// TIA Portal V16 export
// export: Created 2023-03-29T11:03:24.7291018Z, ExportSetting WithDefaults, DisplayName Totally Integrated Automation Portal, DisplayVersion V16 Update 6, DisplayName TIA Portal Version Control Interface, DisplayVersion V16 Update 2, DisplayName TIA Portal Openness, DisplayVersion V16 Update 6, DisplayName STEP 7 Professional, DisplayVersion V16 Update 6, DisplayName STEP 7 Safety, DisplayVersion V16, DisplayName WinCC Advanced, DisplayVersion V16 Update 6
FUNCTION_BLOCK "Client_ModbusTCP_sending_analogs"   // FB4, LAD
TITLE = Wysyłanie analogów
{ S7_Optimized_Access := 'TRUE' }
AUTHOR : rtecmer
VERSION : 0.1
// Wysyłanie pomiarów
// stored: AutoNumber true, IsIECCheckEnabled false, IsRetainMemResEnabled false, MemoryReserve 250, SetENOAutomatically false, UDAEnableTagReadback false
   VAR_IN_OUT
      modbustcp_przetwarzanie_in : Bool;
      modbustcp_przetwarzanie_out : Bool;
   END_VAR
   VAR_TEMP   // added for the SCL form of the ladder/FBD networks
      _w1 : Bool;
      _w2 : Bool;
   END_VAR
BEGIN

REGION Network 2: Inicjacja modbus po błędzie i restarcie
END_REGION

REGION Network 3
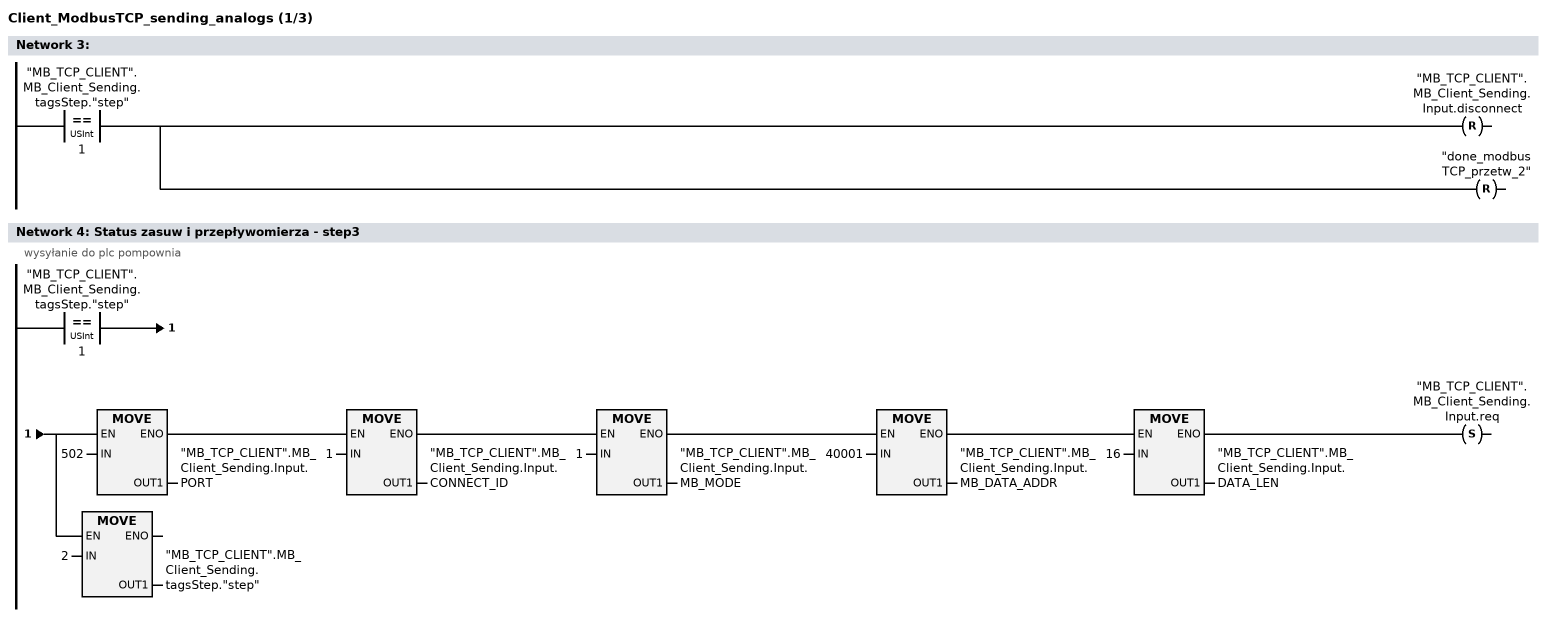
   RUNG wire#powerrail
      { S7_Templates := "SrcType := USInt" } EQ_Contact(in1 := "MB_TCP_CLIENT".MB_Client_Sending.tagsStep."step", in2 := 1)
      wire#w1
      R_Coil( "MB_TCP_CLIENT".MB_Client_Sending.Input.disconnect )
   END_RUNG
   RUNG wire#w1
      R_Coil( "done_modbusTCP_przetw_2" )
   END_RUNG
   // the same network as SCL:
   IF "MB_TCP_CLIENT".MB_Client_Sending.tagsStep."step" = 1 THEN
       "MB_TCP_CLIENT".MB_Client_Sending.Input.disconnect := FALSE;
       "done_modbusTCP_przetw_2" := FALSE;
   END_IF;
END_REGION

REGION Network 4: Status zasuw i przepływomierza - step3
   // wysyłanie do plc pompownia
   RUNG wire#powerrail
      { S7_Templates := "SrcType := USInt" } EQ_Contact(in1 := "MB_TCP_CLIENT".MB_Client_Sending.tagsStep."step", in2 := 1)
      wire#w1
      { S7_GenerateENO := "TRUE" } Move(in := 502, out1 => "MB_TCP_CLIENT".MB_Client_Sending.Input.PORT)
      { S7_GenerateENO := "TRUE" } Move(in := 1, out1 => "MB_TCP_CLIENT".MB_Client_Sending.Input.CONNECT_ID)
      { S7_GenerateENO := "TRUE" } Move(in := 1, out1 => "MB_TCP_CLIENT".MB_Client_Sending.Input.MB_MODE)
      { S7_GenerateENO := "TRUE" } Move(in := 40001, out1 => "MB_TCP_CLIENT".MB_Client_Sending.Input.MB_DATA_ADDR)
      { S7_GenerateENO := "TRUE" } Move(in := 16, out1 => "MB_TCP_CLIENT".MB_Client_Sending.Input.DATA_LEN)
      S_Coil( "MB_TCP_CLIENT".MB_Client_Sending.Input.req )
   END_RUNG
   RUNG wire#w1
      { S7_GenerateENO := "TRUE" } Move(in := 2, out1 => "MB_TCP_CLIENT".MB_Client_Sending.tagsStep."step")
   END_RUNG
   // the same network as SCL:
   // ENO of a box is taken as its EN; it also drops when the box reports an error
   IF "MB_TCP_CLIENT".MB_Client_Sending.tagsStep."step" = 1 THEN
       "MB_TCP_CLIENT".MB_Client_Sending.Input.PORT := 502;
       "MB_TCP_CLIENT".MB_Client_Sending.Input.CONNECT_ID := 1;
       "MB_TCP_CLIENT".MB_Client_Sending.Input.MB_MODE := 1;
       "MB_TCP_CLIENT".MB_Client_Sending.Input.MB_DATA_ADDR := 40001;
       "MB_TCP_CLIENT".MB_Client_Sending.Input.DATA_LEN := 16;
       "MB_TCP_CLIENT".MB_Client_Sending.Input.req := TRUE;
       "MB_TCP_CLIENT".MB_Client_Sending.tagsStep."step" := 2;
   END_IF;
END_REGION

REGION Network 5: step 3
   // Analogi
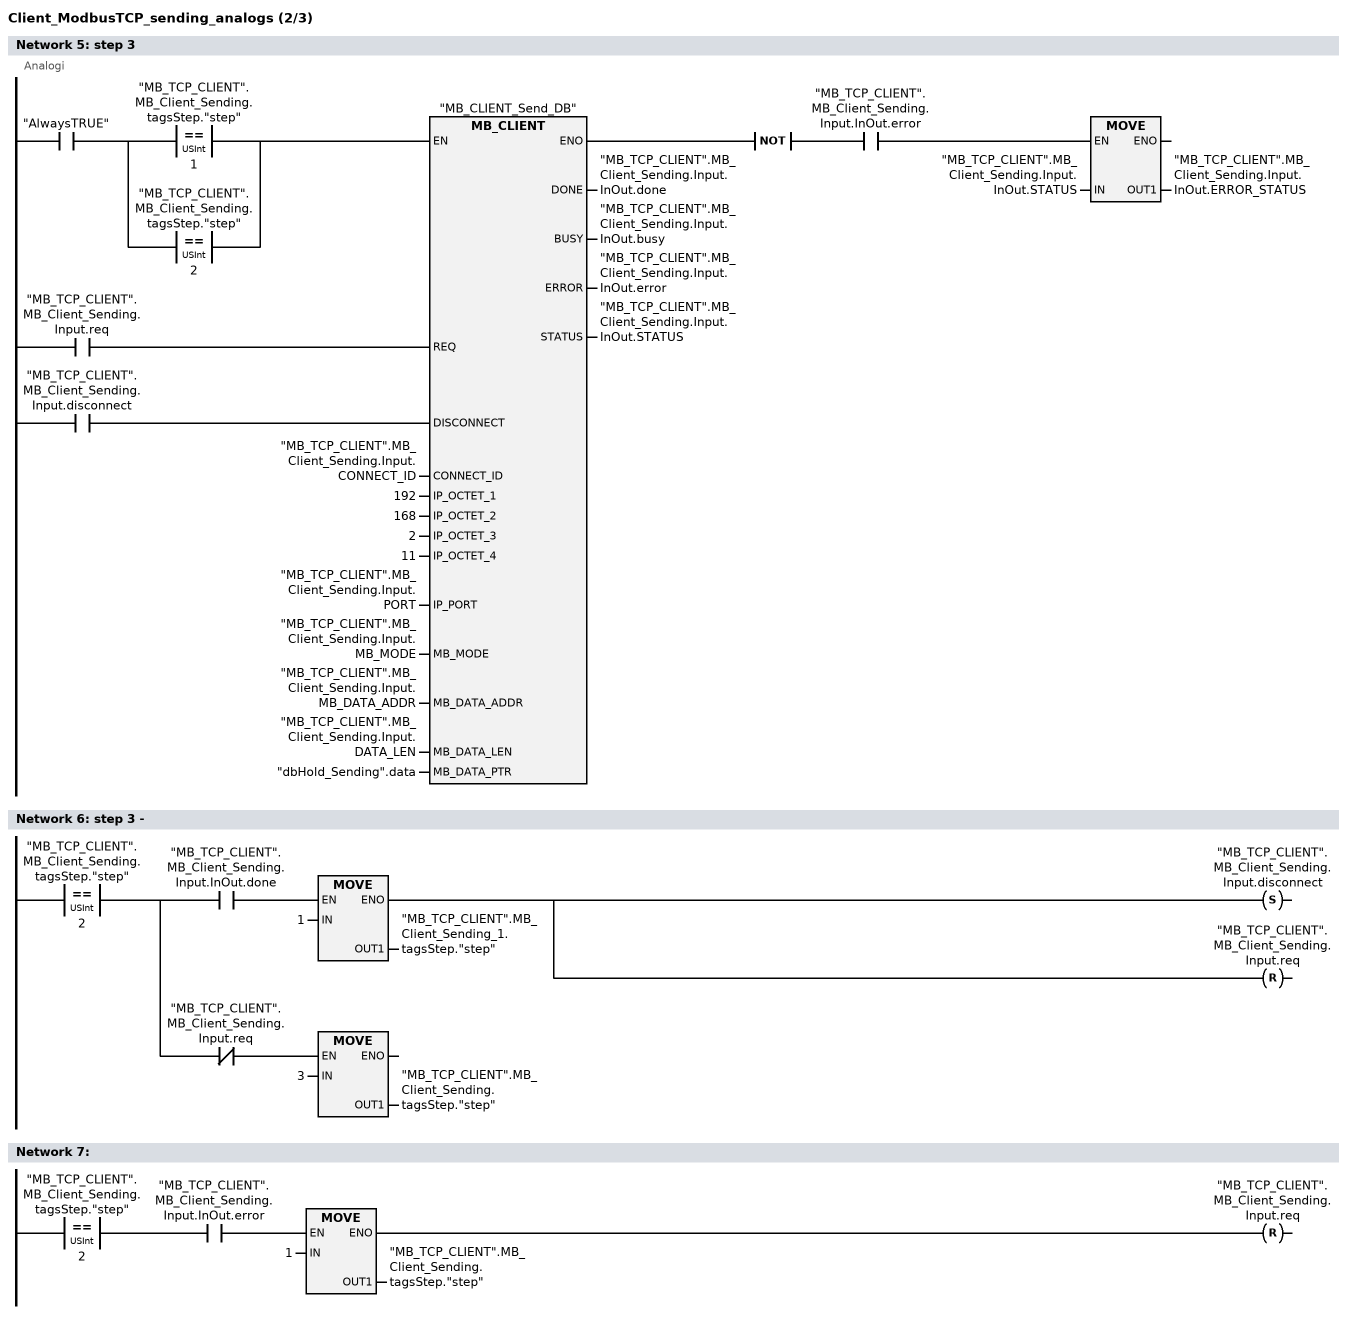
   RUNG wire#powerrail
      Contact( "AlwaysTRUE" )
      wire#w1
      { S7_Templates := "SrcType := USInt" } EQ_Contact(in1 := "MB_TCP_CLIENT".MB_Client_Sending.tagsStep."step", in2 := 1)
      wire#w2
      { S7_Templates := "[card1200 := 1, card1500 := 0]" } "MB_CLIENT_Send_DB".MB_CLIENT(REQ := wire#w3, DISCONNECT := wire#w4, CONNECT_ID := "MB_TCP_CLIENT".MB_Client_Sending.Input.CONNECT_ID, IP_OCTET_1 := 192, IP_OCTET_2 := 168, IP_OCTET_3 := 2, IP_OCTET_4 := 11, IP_PORT := "MB_TCP_CLIENT".MB_Client_Sending.Input.PORT, MB_MODE := "MB_TCP_CLIENT".MB_Client_Sending.Input.MB_MODE, MB_DATA_ADDR := "MB_TCP_CLIENT".MB_Client_Sending.Input.MB_DATA_ADDR, MB_DATA_LEN := "MB_TCP_CLIENT".MB_Client_Sending.Input.DATA_LEN, MB_DATA_PTR := "dbHold_Sending".data, DONE => "MB_TCP_CLIENT".MB_Client_Sending.Input.InOut.done, BUSY => "MB_TCP_CLIENT".MB_Client_Sending.Input.InOut.busy, ERROR => "MB_TCP_CLIENT".MB_Client_Sending.Input.InOut.error, STATUS => "MB_TCP_CLIENT".MB_Client_Sending.Input.InOut.STATUS)
      Not()
      Contact( "MB_TCP_CLIENT".MB_Client_Sending.Input.InOut.error )
      Move(in := "MB_TCP_CLIENT".MB_Client_Sending.Input.InOut.STATUS, out1 => "MB_TCP_CLIENT".MB_Client_Sending.Input.InOut.ERROR_STATUS)
   END_RUNG
   RUNG wire#w1
      { S7_Templates := "SrcType := USInt" } EQ_Contact(in1 := "MB_TCP_CLIENT".MB_Client_Sending.tagsStep."step", in2 := 2)
   END_RUNG wire#w2
   RUNG wire#powerrail
      Contact( "MB_TCP_CLIENT".MB_Client_Sending.Input.req )
   END_RUNG wire#w3
   RUNG wire#powerrail
      Contact( "MB_TCP_CLIENT".MB_Client_Sending.Input.disconnect )
   END_RUNG wire#w4
   // the same network as SCL:
   #_w1 := "AlwaysTRUE" AND (("MB_TCP_CLIENT".MB_Client_Sending.tagsStep."step" = 1) OR ("MB_TCP_CLIENT".MB_Client_Sending.tagsStep."step" = 2));
   "MB_CLIENT_Send_DB"(EN := #_w1,   // MB_CLIENT
                       REQ := "MB_TCP_CLIENT".MB_Client_Sending.Input.req,
                       DISCONNECT := "MB_TCP_CLIENT".MB_Client_Sending.Input.disconnect,
                       CONNECT_ID := "MB_TCP_CLIENT".MB_Client_Sending.Input.CONNECT_ID,
                       IP_OCTET_1 := 192,
                       IP_OCTET_2 := 168,
                       IP_OCTET_3 := 2,
                       IP_OCTET_4 := 11,
                       IP_PORT := "MB_TCP_CLIENT".MB_Client_Sending.Input.PORT,
                       MB_MODE := "MB_TCP_CLIENT".MB_Client_Sending.Input.MB_MODE,
                       MB_DATA_ADDR := "MB_TCP_CLIENT".MB_Client_Sending.Input.MB_DATA_ADDR,
                       MB_DATA_LEN := "MB_TCP_CLIENT".MB_Client_Sending.Input.DATA_LEN,
                       MB_DATA_PTR := "dbHold_Sending".data,
                       DONE => "MB_TCP_CLIENT".MB_Client_Sending.Input.InOut.done,
                       BUSY => "MB_TCP_CLIENT".MB_Client_Sending.Input.InOut.busy,
                       ERROR => "MB_TCP_CLIENT".MB_Client_Sending.Input.InOut.error,
                       STATUS => "MB_TCP_CLIENT".MB_Client_Sending.Input.InOut.STATUS,
                       ENO => #_w2);
   IF NOT #_w2 AND "MB_TCP_CLIENT".MB_Client_Sending.Input.InOut.error THEN
       "MB_TCP_CLIENT".MB_Client_Sending.Input.InOut.ERROR_STATUS := "MB_TCP_CLIENT".MB_Client_Sending.Input.InOut.STATUS;
   END_IF;
END_REGION

REGION Network 6: step 3 -
   RUNG wire#powerrail
      { S7_Templates := "SrcType := USInt" } EQ_Contact(in1 := "MB_TCP_CLIENT".MB_Client_Sending.tagsStep."step", in2 := 2)
      wire#w1
      Contact( "MB_TCP_CLIENT".MB_Client_Sending.Input.InOut.done )
      Move(in := 1, out1 => "MB_TCP_CLIENT".MB_Client_Sending_1.tagsStep."step")
      wire#w2
      S_Coil( "MB_TCP_CLIENT".MB_Client_Sending.Input.disconnect )
   END_RUNG
   RUNG wire#w2
      R_Coil( "MB_TCP_CLIENT".MB_Client_Sending.Input.req )
   END_RUNG
   RUNG wire#w1
      I_Contact( "MB_TCP_CLIENT".MB_Client_Sending.Input.req )
      Move(in := 3, out1 => "MB_TCP_CLIENT".MB_Client_Sending.tagsStep."step")
   END_RUNG
   // the same network as SCL:
   #_w1 := "MB_TCP_CLIENT".MB_Client_Sending.tagsStep."step" = 2;
   IF #_w1 AND "MB_TCP_CLIENT".MB_Client_Sending.Input.InOut.done THEN
       "MB_TCP_CLIENT".MB_Client_Sending_1.tagsStep."step" := 1;
       "MB_TCP_CLIENT".MB_Client_Sending.Input.disconnect := TRUE;
       "MB_TCP_CLIENT".MB_Client_Sending.Input.req := FALSE;
   END_IF;
   IF #_w1 AND NOT "MB_TCP_CLIENT".MB_Client_Sending.Input.req THEN
       "MB_TCP_CLIENT".MB_Client_Sending.tagsStep."step" := 3;
   END_IF;
END_REGION

REGION Network 7
   RUNG wire#powerrail
      { S7_Templates := "SrcType := USInt" } EQ_Contact(in1 := "MB_TCP_CLIENT".MB_Client_Sending.tagsStep."step", in2 := 2)
      Contact( "MB_TCP_CLIENT".MB_Client_Sending.Input.InOut.error )
      Move(in := 1, out1 => "MB_TCP_CLIENT".MB_Client_Sending.tagsStep."step")
      R_Coil( "MB_TCP_CLIENT".MB_Client_Sending.Input.req )
   END_RUNG
   // the same network as SCL:
   #_w1 := ("MB_TCP_CLIENT".MB_Client_Sending.tagsStep."step" = 2) AND "MB_TCP_CLIENT".MB_Client_Sending.Input.InOut.error;
   IF #_w1 THEN
       "MB_TCP_CLIENT".MB_Client_Sending.tagsStep."step" := 1;
       "MB_TCP_CLIENT".MB_Client_Sending.Input.req := FALSE;
   END_IF;
END_REGION

REGION Network 8
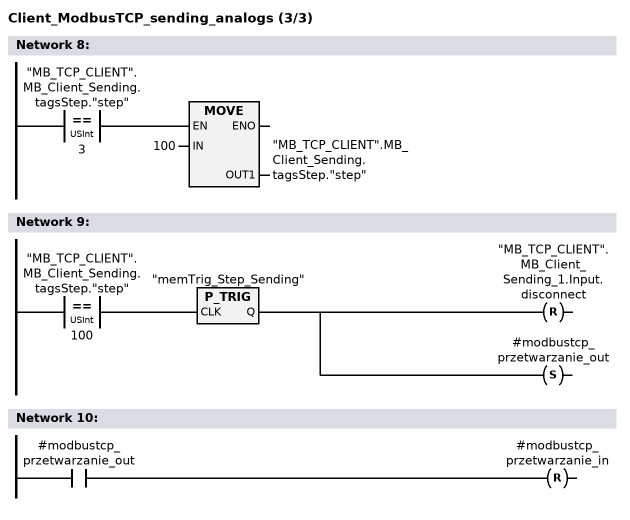
   RUNG wire#powerrail
      { S7_Templates := "SrcType := USInt" } EQ_Contact(in1 := "MB_TCP_CLIENT".MB_Client_Sending.tagsStep."step", in2 := 3)
      Move(in := 100, out1 => "MB_TCP_CLIENT".MB_Client_Sending.tagsStep."step")
   END_RUNG
   // the same network as SCL:
   IF "MB_TCP_CLIENT".MB_Client_Sending.tagsStep."step" = 3 THEN
       "MB_TCP_CLIENT".MB_Client_Sending.tagsStep."step" := 100;
   END_IF;
END_REGION

REGION Network 9
   RUNG wire#powerrail
      { S7_Templates := "SrcType := USInt" } EQ_Contact(in1 := "MB_TCP_CLIENT".MB_Client_Sending.tagsStep."step", in2 := 100)
      P_Trig( "memTrig_Step_Sending" )
      wire#w1
      R_Coil( "MB_TCP_CLIENT".MB_Client_Sending_1.Input.disconnect )
   END_RUNG
   RUNG wire#w1
      S_Coil( #modbustcp_przetwarzanie_out )
   END_RUNG
   // the same network as SCL:
   #_w1 := "MB_TCP_CLIENT".MB_Client_Sending.tagsStep."step" = 100;
   #_w2 := #_w1 AND NOT "memTrig_Step_Sending";   // rising edge
   "memTrig_Step_Sending" := #_w1;
   IF #_w2 THEN
       "MB_TCP_CLIENT".MB_Client_Sending_1.Input.disconnect := FALSE;
       #modbustcp_przetwarzanie_out := TRUE;
   END_IF;
END_REGION

REGION Network 10
   RUNG wire#powerrail
      Contact( #modbustcp_przetwarzanie_out )
      R_Coil( #modbustcp_przetwarzanie_in )
   END_RUNG
   // the same network as SCL:
   IF #modbustcp_przetwarzanie_out THEN #modbustcp_przetwarzanie_in := FALSE; END_IF;
END_REGION
END_FUNCTION_BLOCK
